{attribute 'GeneratedUsingTerminal: EK1100-0000-0018'}
{attribute addProperty BoxType "EK1100-0000-0018"}
{attribute addProperty Id "Beckhoff_EL1xxxEK1122Beckhoff_EL1xxxEK1122_A32C991B2A_0001_EL1002_0000_0000EL1002_90CA79196A_0002_EL1002_0000_0016EL1002_90CA79196A_0003_EL1002_0000_0017EL1002_90CA79196A_0004_EL1002_0000_0018EL1002_90CA79196A_0005_EL1004_0000_0000EL1004_BF8C6BFA8A_0006_EL1004_0000_0016EL1004_BF8C6BFA8A_0007_EL1004_0000_0017EL1004_BF8C6BFA8A_0008_EL1004_0000_0018EL1004_BF8C6BFA8A_0009_EL1004_0000_0019EL1004_BF8C6BFA8A_0010_EL1004_0010_0000EL1004_BF8C6BFA8A_0011_EL1004_0010_0016EL1004_BF8C6BFA8A_0012_EL1004_0010_0017EL1004_BF8C6BFA8A_0013_EL1004_0010_0018EL1004_BF8C6BFA8A_0014_EL1004_0020_0016EL1004_BF8C6BFA8A_0015_EL1008_0000_0016EL1008_4201D0AB12A_0016_EL1008_0000_0017EL1008_4201D0AB12A_0017_EL1008_0000_0018EL1008_4201D0AB12A_0018_EL1012_0000_0000EL1012_90CA79196A_0019_EL1012_0000_0016EL1012_90CA79196A_0020_EL1012_0000_0017EL1012_90CA79196A_0021_EL1012_0000_0018EL1012_90CA79196A_0022_EL1014_0000_0000EL1014_BF8C6BFA8A_0023_EL1014_0000_0016EL1014_BF8C6BFA8A_0024_EL1014_0000_0017EL1014_BF8C6BFA8A_0025_EL1014_0000_0018EL1014_BF8C6BFA8A_0026_EL1014_0000_0019EL1014_BF8C6BFA8A_0027_EL1014_0010_0000EL1014_BF8C6BFA8A_0028_EL1014_0010_0016EL1014_BF8C6BFA8A_0029_EL1014_0010_0017EL1014_BF8C6BFA8A_0030_EL1014_0010_0018EL1014_BF8C6BFA8A_0031_EL1014_0010_0019EL1014_BF8C6BFA8A_0032_EL1018_0000_0016EL1018_4201D0AB12A_0033_EL1018_0000_0017EL1018_4201D0AB12A_0034_EL1018_0000_0018EL1018_4201D0AB12A_0035_EL1024_0000_0016EL1024_BF8C6BFA8A_0036_EL1024_0000_0017EL1024_BF8C6BFA8A_0037_EL1024_0000_0018EL1024_BF8C6BFA8A_0038_EL1034_0000_0016EL1034_BF8C6BFA8A_0039_EL1034_0000_0017EL1034_BF8C6BFA8A_0040_EL1034_0000_0018EL1034_BF8C6BFA8A_0041_EL1052_0000_0016EL1052_FE4CEFB88A_0042_EL1054_0000_0016EL1054_5971E93D12A_0043_EL1084_0000_0016EL1084_BF8C6BFA8A_0044_EL1084_0000_0017EL1084_BF8C6BFA8A_0045_EL1084_0000_0018EL1084_BF8C6BFA8A_0046_EL1088_0000_0016EL1088_4201D0AB12A_0047_EL1088_0000_0017EL1088_4201D0AB12A_0048_EL1088_0000_0018EL1088_4201D0AB12A_0049_EL1094_0000_0016EL1094_BF8C6BFA8A_0050_EL1094_0000_0017EL1094_BF8C6BFA8A_0051_EL1094_0000_0018EL1094_BF8C6BFA8A_0052_EL1098_0000_0016EL1098_4201D0AB12A_0053_EL1098_0000_0017EL1098_4201D0AB12A_0054_EL1098_0000_0018EL1098_4201D0AB12A_0055_EL1104_0000_0016EL1104_BF8C6BFA8A_0056_EL1104_0000_0017EL1104_BF8C6BFA8A_0057_EL1104_0000_0018EL1104_BF8C6BFA8A_0058_EL1114_0000_0016EL1114_BF8C6BFA8A_0059_EL1114_0000_0017EL1114_BF8C6BFA8A_0060_EL1114_0000_0018EL1114_BF8C6BFA8A_0061_EL1124_0000_0016EL1124_BF8C6BFA8A_0062_EL1124_0000_0017EL1124_BF8C6BFA8A_0063_EL1124_0000_0018EL1124_BF8C6BFA8A_0064_EL1134_0000_0016EL1134_BF8C6BFA8A_0065_EL1134_0000_0017EL1134_BF8C6BFA8A_0066_EL1134_0000_0018EL1134_BF8C6BFA8A_0067_EL1144_0000_0016EL1144_BF8C6BFA8A_0068_EL1144_0000_0017EL1144_BF8C6BFA8A_0069_EL1144_0000_0018EL1144_BF8C6BFA8A_0070_EL1202_0000_0016EL1202_90CA79196A_0071_EL1202_0000_0017EL1202_90CA79196A_0072_EL1202_0000_0018EL1202_90CA79196A_0073_EL1202_0000_0019EL1202_90CA79196A_0074_EL1202_0100_0016EL1202_5869074F22A_0075_EL1202_0100_0017EL1202_5869074F22A_0076_EL1202_0100_0018EL1202_5869074F22A_0077_EL1202_0100_0019EL1202_5869074F22A_0078_EL1252_0000_0017EL1252_F879009148A_0079_EL1252_0000_0018EL1252_671E5FD948A_0080_EL1252_0000_0019EL1252_671E5FD948A_0081_EL1252_0000_0020EL1252_671E5FD948A_0082_EL1252_0000_0021EL1252_671E5FD948A_0083_EL1252_0000_0022EL1252_671E5FD948A_0084_EL1252_0010_0019EL1252_671E5FD948A_0085_EL1252_0010_0020EL1252_671E5FD948A_0086_EL1252_0010_0021EL1252_671E5FD948A_0087_EL1252_0050_0016EL1252_671E5FD948A_0088_EL1252_0050_0017EL1252_671E5FD948A_0089_EL1252_0050_0018EL1252_671E5FD948A_0090_EL1254_0000_0000EL1254_F2A8C39584A_0091_EL1262_0000_0002EL1262_BA5C56E540A_0092_EL1262_0000_0003EL1262_BA5C56E540A_0093_EL1262_0050_0002EL1262_BA5C56E540A_0094_EL1262_0050_0003EL1262_BA5C56E540A_0095_EL1258_0000_0016EL1258_D4F4E2D7484A_0096_EL1258_0000_0017EL1258_D4F4E2D7484A_0097_EL1258_0010_0017EL1258_FEC2AC79124A_0098_EL1259_0000_0016EL1259_C8DF9E9D972A_0099_EL1259_0000_0017EL1259_32A74CEC980A_0100_EL1259_0000_0018EL1259_32A74CEC980A_0101_EL1382_0000_0016EL1382_FE4CEFB88A_0102_EL1382_0000_0017EL1382_FE4CEFB88A_0103_EL1382_0000_0018EL1382_FE4CEFB88A_0104_EL1702_0000_0016EL1702_90CA79196A_0105_EL1702_0000_0017EL1702_90CA79196A_0106_EL1702_0020_0016EL1702_90CA79196A_0107_EL1712_0000_0016EL1712_90CA79196A_0108_EL1712_0020_0016EL1712_90CA79196A_0109_EL1722_0000_0016EL1722_90CA79196A_0110_EL1722_0000_0017EL1722_90CA79196A_0111_EL1804_0000_0016EL1804_BF8C6BFA8A_0112_EL1804_0000_0017EL1804_BF8C6BFA8A_0113_EL1804_0000_0018EL1804_BF8C6BFA8A_0114_EL1808_0000_0016EL1808_4201D0AB12A_0115_EL1808_0000_0017EL1808_4201D0AB12A_0116_EL1808_0000_0018EL1808_4201D0AB12A_0117_EL1809_0000_0016EL1809_FD7895E220A_0118_EL1809_0000_0017EL1809_FD7895E220A_0119_EL1809_0000_0018EL1809_FD7895E220A_0120_EL1814_0000_0016EL1814_BF8C6BFA8A_0121_EL1814_0000_0017EL1814_BF8C6BFA8A_0122_EL1814_0000_0018EL1814_BF8C6BFA8A_0123_EL1819_0000_0016EL1819_FD7895E220A_0124_EL1819_0000_0017EL1819_FD7895E220A_0125_EL1819_0000_0018EL1819_FD7895E220A_0126_EL1852_0000_0016EL1852_B9F455E920A_0127_EL1859_0000_0016EL1859_B9F455E920A_0128_EL1859_0000_0017EL1859_B9F455E920A_0129_EL1859_0000_0018EL1859_B9F455E920A_0130_EL1862_0000_0016EL1862_FD7895E220A_0131_EL1862_0000_0017EL1862_FD7895E220A_0132_EL1862_0000_0018EL1862_FD7895E220A_0133_EL1862_0000_0019EL1862_FD7895E220A_0134_EL1862_0010_0016EL1862_FD7895E220A_0135_EL1862_0010_0017EL1862_FD7895E220A_0136_EL1862_0010_0018EL1862_FD7895E220A_0137_EL1862_0010_0019EL1862_FD7895E220A_0138_EL1872_0000_0016EL1872_FD7895E220A_0139_EL1872_0000_0017EL1872_FD7895E220A_0140_EL1872_0000_0018EL1872_FD7895E220A_0141_EL1872_0010_0016EL1872_FD7895E220A_0142_EL1889_0000_0016EL1889_FD7895E220A_0143_EL1889_0000_0017EL1889_FD7895E220A_0144_EL1889_0000_0018EL1889_FD7895E220A_0145_EL1889_0000_0019EL1889_FD7895E220A_0146_EL1899_0000_0016EL1899_FD7895E220"}
{attribute addProperty CRC "3910229889"}
{attribute addProperty Size "6236"}
TYPE Beckhoff_EL1xxx_E9115F81 EXTENDS EK1100_AB5A9467 :
STRUCT
	{attribute addProperty Name "Beckhoff_EL1xxxEK1122"}
	Beckhoff_EL1xxxEK1122 : Beckhoff_EL1xxxEK1122_A32C991B;
	{attribute addProperty Name "A_0001_EL1002_0000_0000"}
	A_0001_EL1002_0000_0000 : EL1002_90CA7919;
	{attribute addProperty Name "A_0002_EL1002_0000_0016"}
	A_0002_EL1002_0000_0016 : EL1002_90CA7919;
	{attribute addProperty Name "A_0003_EL1002_0000_0017"}
	A_0003_EL1002_0000_0017 : EL1002_90CA7919;
	{attribute addProperty Name "A_0004_EL1002_0000_0018"}
	A_0004_EL1002_0000_0018 : EL1002_90CA7919;
	{attribute addProperty Name "A_0005_EL1004_0000_0000"}
	A_0005_EL1004_0000_0000 : EL1004_BF8C6BFA;
	{attribute addProperty Name "A_0006_EL1004_0000_0016"}
	A_0006_EL1004_0000_0016 : EL1004_BF8C6BFA;
	{attribute addProperty Name "A_0007_EL1004_0000_0017"}
	A_0007_EL1004_0000_0017 : EL1004_BF8C6BFA;
	{attribute addProperty Name "A_0008_EL1004_0000_0018"}
	A_0008_EL1004_0000_0018 : EL1004_BF8C6BFA;
	{attribute addProperty Name "A_0009_EL1004_0000_0019"}
	A_0009_EL1004_0000_0019 : EL1004_BF8C6BFA;
	{attribute addProperty Name "A_0010_EL1004_0010_0000"}
	A_0010_EL1004_0010_0000 : EL1004_BF8C6BFA;
	{attribute addProperty Name "A_0011_EL1004_0010_0016"}
	A_0011_EL1004_0010_0016 : EL1004_BF8C6BFA;
	{attribute addProperty Name "A_0012_EL1004_0010_0017"}
	A_0012_EL1004_0010_0017 : EL1004_BF8C6BFA;
	{attribute addProperty Name "A_0013_EL1004_0010_0018"}
	A_0013_EL1004_0010_0018 : EL1004_BF8C6BFA;
	{attribute addProperty Name "A_0014_EL1004_0020_0016"}
	A_0014_EL1004_0020_0016 : EL1004_BF8C6BFA;
	{attribute addProperty Name "A_0015_EL1008_0000_0016"}
	A_0015_EL1008_0000_0016 : EL1008_4201D0AB;
	{attribute addProperty Name "A_0016_EL1008_0000_0017"}
	A_0016_EL1008_0000_0017 : EL1008_4201D0AB;
	{attribute addProperty Name "A_0017_EL1008_0000_0018"}
	A_0017_EL1008_0000_0018 : EL1008_4201D0AB;
	{attribute addProperty Name "A_0018_EL1012_0000_0000"}
	A_0018_EL1012_0000_0000 : EL1012_90CA7919;
	{attribute addProperty Name "A_0019_EL1012_0000_0016"}
	A_0019_EL1012_0000_0016 : EL1012_90CA7919;
	{attribute addProperty Name "A_0020_EL1012_0000_0017"}
	A_0020_EL1012_0000_0017 : EL1012_90CA7919;
	{attribute addProperty Name "A_0021_EL1012_0000_0018"}
	A_0021_EL1012_0000_0018 : EL1012_90CA7919;
	{attribute addProperty Name "A_0022_EL1014_0000_0000"}
	A_0022_EL1014_0000_0000 : EL1014_BF8C6BFA;
	{attribute addProperty Name "A_0023_EL1014_0000_0016"}
	A_0023_EL1014_0000_0016 : EL1014_BF8C6BFA;
	{attribute addProperty Name "A_0024_EL1014_0000_0017"}
	A_0024_EL1014_0000_0017 : EL1014_BF8C6BFA;
	{attribute addProperty Name "A_0025_EL1014_0000_0018"}
	A_0025_EL1014_0000_0018 : EL1014_BF8C6BFA;
	{attribute addProperty Name "A_0026_EL1014_0000_0019"}
	A_0026_EL1014_0000_0019 : EL1014_BF8C6BFA;
	{attribute addProperty Name "A_0027_EL1014_0010_0000"}
	A_0027_EL1014_0010_0000 : EL1014_BF8C6BFA;
	{attribute addProperty Name "A_0028_EL1014_0010_0016"}
	A_0028_EL1014_0010_0016 : EL1014_BF8C6BFA;
	{attribute addProperty Name "A_0029_EL1014_0010_0017"}
	A_0029_EL1014_0010_0017 : EL1014_BF8C6BFA;
	{attribute addProperty Name "A_0030_EL1014_0010_0018"}
	A_0030_EL1014_0010_0018 : EL1014_BF8C6BFA;
	{attribute addProperty Name "A_0031_EL1014_0010_0019"}
	A_0031_EL1014_0010_0019 : EL1014_BF8C6BFA;
	{attribute addProperty Name "A_0032_EL1018_0000_0016"}
	A_0032_EL1018_0000_0016 : EL1018_4201D0AB;
	{attribute addProperty Name "A_0033_EL1018_0000_0017"}
	A_0033_EL1018_0000_0017 : EL1018_4201D0AB;
	{attribute addProperty Name "A_0034_EL1018_0000_0018"}
	A_0034_EL1018_0000_0018 : EL1018_4201D0AB;
	{attribute addProperty Name "A_0035_EL1024_0000_0016"}
	A_0035_EL1024_0000_0016 : EL1024_BF8C6BFA;
	{attribute addProperty Name "A_0036_EL1024_0000_0017"}
	A_0036_EL1024_0000_0017 : EL1024_BF8C6BFA;
	{attribute addProperty Name "A_0037_EL1024_0000_0018"}
	A_0037_EL1024_0000_0018 : EL1024_BF8C6BFA;
	{attribute addProperty Name "A_0038_EL1034_0000_0016"}
	A_0038_EL1034_0000_0016 : EL1034_BF8C6BFA;
	{attribute addProperty Name "A_0039_EL1034_0000_0017"}
	A_0039_EL1034_0000_0017 : EL1034_BF8C6BFA;
	{attribute addProperty Name "A_0040_EL1034_0000_0018"}
	A_0040_EL1034_0000_0018 : EL1034_BF8C6BFA;
	{attribute addProperty Name "A_0041_EL1052_0000_0016"}
	A_0041_EL1052_0000_0016 : EL1052_FE4CEFB8;
	{attribute addProperty Name "A_0042_EL1054_0000_0016"}
	A_0042_EL1054_0000_0016 : EL1054_5971E93D;
	{attribute addProperty Name "A_0043_EL1084_0000_0016"}
	A_0043_EL1084_0000_0016 : EL1084_BF8C6BFA;
	{attribute addProperty Name "A_0044_EL1084_0000_0017"}
	A_0044_EL1084_0000_0017 : EL1084_BF8C6BFA;
	{attribute addProperty Name "A_0045_EL1084_0000_0018"}
	A_0045_EL1084_0000_0018 : EL1084_BF8C6BFA;
	{attribute addProperty Name "A_0046_EL1088_0000_0016"}
	A_0046_EL1088_0000_0016 : EL1088_4201D0AB;
	{attribute addProperty Name "A_0047_EL1088_0000_0017"}
	A_0047_EL1088_0000_0017 : EL1088_4201D0AB;
	{attribute addProperty Name "A_0048_EL1088_0000_0018"}
	A_0048_EL1088_0000_0018 : EL1088_4201D0AB;
	{attribute addProperty Name "A_0049_EL1094_0000_0016"}
	A_0049_EL1094_0000_0016 : EL1094_BF8C6BFA;
	{attribute addProperty Name "A_0050_EL1094_0000_0017"}
	A_0050_EL1094_0000_0017 : EL1094_BF8C6BFA;
	{attribute addProperty Name "A_0051_EL1094_0000_0018"}
	A_0051_EL1094_0000_0018 : EL1094_BF8C6BFA;
	{attribute addProperty Name "A_0052_EL1098_0000_0016"}
	A_0052_EL1098_0000_0016 : EL1098_4201D0AB;
	{attribute addProperty Name "A_0053_EL1098_0000_0017"}
	A_0053_EL1098_0000_0017 : EL1098_4201D0AB;
	{attribute addProperty Name "A_0054_EL1098_0000_0018"}
	A_0054_EL1098_0000_0018 : EL1098_4201D0AB;
	{attribute addProperty Name "A_0055_EL1104_0000_0016"}
	A_0055_EL1104_0000_0016 : EL1104_BF8C6BFA;
	{attribute addProperty Name "A_0056_EL1104_0000_0017"}
	A_0056_EL1104_0000_0017 : EL1104_BF8C6BFA;
	{attribute addProperty Name "A_0057_EL1104_0000_0018"}
	A_0057_EL1104_0000_0018 : EL1104_BF8C6BFA;
	{attribute addProperty Name "A_0058_EL1114_0000_0016"}
	A_0058_EL1114_0000_0016 : EL1114_BF8C6BFA;
	{attribute addProperty Name "A_0059_EL1114_0000_0017"}
	A_0059_EL1114_0000_0017 : EL1114_BF8C6BFA;
	{attribute addProperty Name "A_0060_EL1114_0000_0018"}
	A_0060_EL1114_0000_0018 : EL1114_BF8C6BFA;
	{attribute addProperty Name "A_0061_EL1124_0000_0016"}
	A_0061_EL1124_0000_0016 : EL1124_BF8C6BFA;
	{attribute addProperty Name "A_0062_EL1124_0000_0017"}
	A_0062_EL1124_0000_0017 : EL1124_BF8C6BFA;
	{attribute addProperty Name "A_0063_EL1124_0000_0018"}
	A_0063_EL1124_0000_0018 : EL1124_BF8C6BFA;
	{attribute addProperty Name "A_0064_EL1134_0000_0016"}
	A_0064_EL1134_0000_0016 : EL1134_BF8C6BFA;
	{attribute addProperty Name "A_0065_EL1134_0000_0017"}
	A_0065_EL1134_0000_0017 : EL1134_BF8C6BFA;
	{attribute addProperty Name "A_0066_EL1134_0000_0018"}
	A_0066_EL1134_0000_0018 : EL1134_BF8C6BFA;
	{attribute addProperty Name "A_0067_EL1144_0000_0016"}
	A_0067_EL1144_0000_0016 : EL1144_BF8C6BFA;
	{attribute addProperty Name "A_0068_EL1144_0000_0017"}
	A_0068_EL1144_0000_0017 : EL1144_BF8C6BFA;
	{attribute addProperty Name "A_0069_EL1144_0000_0018"}
	A_0069_EL1144_0000_0018 : EL1144_BF8C6BFA;
	{attribute addProperty Name "A_0070_EL1202_0000_0016"}
	A_0070_EL1202_0000_0016 : EL1202_90CA7919;
	{attribute addProperty Name "A_0071_EL1202_0000_0017"}
	A_0071_EL1202_0000_0017 : EL1202_90CA7919;
	{attribute addProperty Name "A_0072_EL1202_0000_0018"}
	A_0072_EL1202_0000_0018 : EL1202_90CA7919;
	{attribute addProperty Name "A_0073_EL1202_0000_0019"}
	A_0073_EL1202_0000_0019 : EL1202_90CA7919;
	{attribute addProperty Name "A_0074_EL1202_0100_0016"}
	A_0074_EL1202_0100_0016 : EL1202_5869074F;
	{attribute addProperty Name "A_0075_EL1202_0100_0017"}
	A_0075_EL1202_0100_0017 : EL1202_5869074F;
	{attribute addProperty Name "A_0076_EL1202_0100_0018"}
	A_0076_EL1202_0100_0018 : EL1202_5869074F;
	{attribute addProperty Name "A_0077_EL1202_0100_0019"}
	A_0077_EL1202_0100_0019 : EL1202_5869074F;
	{attribute addProperty Name "A_0078_EL1252_0000_0017"}
	A_0078_EL1252_0000_0017 : EL1252_F8790091;
	{attribute addProperty Name "A_0079_EL1252_0000_0018"}
	A_0079_EL1252_0000_0018 : EL1252_671E5FD9;
	{attribute addProperty Name "A_0080_EL1252_0000_0019"}
	A_0080_EL1252_0000_0019 : EL1252_671E5FD9;
	{attribute addProperty Name "A_0081_EL1252_0000_0020"}
	A_0081_EL1252_0000_0020 : EL1252_671E5FD9;
	{attribute addProperty Name "A_0082_EL1252_0000_0021"}
	A_0082_EL1252_0000_0021 : EL1252_671E5FD9;
	{attribute addProperty Name "A_0083_EL1252_0000_0022"}
	A_0083_EL1252_0000_0022 : EL1252_671E5FD9;
	{attribute addProperty Name "A_0084_EL1252_0010_0019"}
	A_0084_EL1252_0010_0019 : EL1252_671E5FD9;
	{attribute addProperty Name "A_0085_EL1252_0010_0020"}
	A_0085_EL1252_0010_0020 : EL1252_671E5FD9;
	{attribute addProperty Name "A_0086_EL1252_0010_0021"}
	A_0086_EL1252_0010_0021 : EL1252_671E5FD9;
	{attribute addProperty Name "A_0087_EL1252_0050_0016"}
	A_0087_EL1252_0050_0016 : EL1252_671E5FD9;
	{attribute addProperty Name "A_0088_EL1252_0050_0017"}
	A_0088_EL1252_0050_0017 : EL1252_671E5FD9;
	{attribute addProperty Name "A_0089_EL1252_0050_0018"}
	A_0089_EL1252_0050_0018 : EL1252_671E5FD9;
	{attribute addProperty Name "A_0090_EL1254_0000_0000"}
	A_0090_EL1254_0000_0000 : EL1254_F2A8C395;
	{attribute addProperty Name "A_0091_EL1262_0000_0002"}
	A_0091_EL1262_0000_0002 : EL1262_BA5C56E5;
	{attribute addProperty Name "A_0092_EL1262_0000_0003"}
	A_0092_EL1262_0000_0003 : EL1262_BA5C56E5;
	{attribute addProperty Name "A_0093_EL1262_0050_0002"}
	A_0093_EL1262_0050_0002 : EL1262_BA5C56E5;
	{attribute addProperty Name "A_0094_EL1262_0050_0003"}
	A_0094_EL1262_0050_0003 : EL1262_BA5C56E5;
	{attribute addProperty Name "A_0095_EL1258_0000_0016"}
	A_0095_EL1258_0000_0016 : EL1258_D4F4E2D7;
	{attribute addProperty Name "A_0096_EL1258_0000_0017"}
	A_0096_EL1258_0000_0017 : EL1258_D4F4E2D7;
	{attribute addProperty Name "A_0097_EL1258_0010_0017"}
	A_0097_EL1258_0010_0017 : EL1258_FEC2AC79;
	{attribute addProperty Name "A_0098_EL1259_0000_0016"}
	A_0098_EL1259_0000_0016 : EL1259_C8DF9E9D;
	{attribute addProperty Name "A_0099_EL1259_0000_0017"}
	A_0099_EL1259_0000_0017 : EL1259_32A74CEC;
	{attribute addProperty Name "A_0100_EL1259_0000_0018"}
	A_0100_EL1259_0000_0018 : EL1259_32A74CEC;
	{attribute addProperty Name "A_0101_EL1382_0000_0016"}
	A_0101_EL1382_0000_0016 : EL1382_FE4CEFB8;
	{attribute addProperty Name "A_0102_EL1382_0000_0017"}
	A_0102_EL1382_0000_0017 : EL1382_FE4CEFB8;
	{attribute addProperty Name "A_0103_EL1382_0000_0018"}
	A_0103_EL1382_0000_0018 : EL1382_FE4CEFB8;
	{attribute addProperty Name "A_0104_EL1702_0000_0016"}
	A_0104_EL1702_0000_0016 : EL1702_90CA7919;
	{attribute addProperty Name "A_0105_EL1702_0000_0017"}
	A_0105_EL1702_0000_0017 : EL1702_90CA7919;
	{attribute addProperty Name "A_0106_EL1702_0020_0016"}
	A_0106_EL1702_0020_0016 : EL1702_90CA7919;
	{attribute addProperty Name "A_0107_EL1712_0000_0016"}
	A_0107_EL1712_0000_0016 : EL1712_90CA7919;
	{attribute addProperty Name "A_0108_EL1712_0020_0016"}
	A_0108_EL1712_0020_0016 : EL1712_90CA7919;
	{attribute addProperty Name "A_0109_EL1722_0000_0016"}
	A_0109_EL1722_0000_0016 : EL1722_90CA7919;
	{attribute addProperty Name "A_0110_EL1722_0000_0017"}
	A_0110_EL1722_0000_0017 : EL1722_90CA7919;
	{attribute addProperty Name "A_0111_EL1804_0000_0016"}
	A_0111_EL1804_0000_0016 : EL1804_BF8C6BFA;
	{attribute addProperty Name "A_0112_EL1804_0000_0017"}
	A_0112_EL1804_0000_0017 : EL1804_BF8C6BFA;
	{attribute addProperty Name "A_0113_EL1804_0000_0018"}
	A_0113_EL1804_0000_0018 : EL1804_BF8C6BFA;
	{attribute addProperty Name "A_0114_EL1808_0000_0016"}
	A_0114_EL1808_0000_0016 : EL1808_4201D0AB;
	{attribute addProperty Name "A_0115_EL1808_0000_0017"}
	A_0115_EL1808_0000_0017 : EL1808_4201D0AB;
	{attribute addProperty Name "A_0116_EL1808_0000_0018"}
	A_0116_EL1808_0000_0018 : EL1808_4201D0AB;
	{attribute addProperty Name "A_0117_EL1809_0000_0016"}
	A_0117_EL1809_0000_0016 : EL1809_FD7895E2;
	{attribute addProperty Name "A_0118_EL1809_0000_0017"}
	A_0118_EL1809_0000_0017 : EL1809_FD7895E2;
	{attribute addProperty Name "A_0119_EL1809_0000_0018"}
	A_0119_EL1809_0000_0018 : EL1809_FD7895E2;
	{attribute addProperty Name "A_0120_EL1814_0000_0016"}
	A_0120_EL1814_0000_0016 : EL1814_BF8C6BFA;
	{attribute addProperty Name "A_0121_EL1814_0000_0017"}
	A_0121_EL1814_0000_0017 : EL1814_BF8C6BFA;
	{attribute addProperty Name "A_0122_EL1814_0000_0018"}
	A_0122_EL1814_0000_0018 : EL1814_BF8C6BFA;
	{attribute addProperty Name "A_0123_EL1819_0000_0016"}
	A_0123_EL1819_0000_0016 : EL1819_FD7895E2;
	{attribute addProperty Name "A_0124_EL1819_0000_0017"}
	A_0124_EL1819_0000_0017 : EL1819_FD7895E2;
	{attribute addProperty Name "A_0125_EL1819_0000_0018"}
	A_0125_EL1819_0000_0018 : EL1819_FD7895E2;
	{attribute addProperty Name "A_0126_EL1852_0000_0016"}
	A_0126_EL1852_0000_0016 : EL1852_B9F455E9;
	{attribute addProperty Name "A_0127_EL1859_0000_0016"}
	A_0127_EL1859_0000_0016 : EL1859_B9F455E9;
	{attribute addProperty Name "A_0128_EL1859_0000_0017"}
	A_0128_EL1859_0000_0017 : EL1859_B9F455E9;
	{attribute addProperty Name "A_0129_EL1859_0000_0018"}
	A_0129_EL1859_0000_0018 : EL1859_B9F455E9;
	{attribute addProperty Name "A_0130_EL1862_0000_0016"}
	A_0130_EL1862_0000_0016 : EL1862_FD7895E2;
	{attribute addProperty Name "A_0131_EL1862_0000_0017"}
	A_0131_EL1862_0000_0017 : EL1862_FD7895E2;
	{attribute addProperty Name "A_0132_EL1862_0000_0018"}
	A_0132_EL1862_0000_0018 : EL1862_FD7895E2;
	{attribute addProperty Name "A_0133_EL1862_0000_0019"}
	A_0133_EL1862_0000_0019 : EL1862_FD7895E2;
	{attribute addProperty Name "A_0134_EL1862_0010_0016"}
	A_0134_EL1862_0010_0016 : EL1862_FD7895E2;
	{attribute addProperty Name "A_0135_EL1862_0010_0017"}
	A_0135_EL1862_0010_0017 : EL1862_FD7895E2;
	{attribute addProperty Name "A_0136_EL1862_0010_0018"}
	A_0136_EL1862_0010_0018 : EL1862_FD7895E2;
	{attribute addProperty Name "A_0137_EL1862_0010_0019"}
	A_0137_EL1862_0010_0019 : EL1862_FD7895E2;
	{attribute addProperty Name "A_0138_EL1872_0000_0016"}
	A_0138_EL1872_0000_0016 : EL1872_FD7895E2;
	{attribute addProperty Name "A_0139_EL1872_0000_0017"}
	A_0139_EL1872_0000_0017 : EL1872_FD7895E2;
	{attribute addProperty Name "A_0140_EL1872_0000_0018"}
	A_0140_EL1872_0000_0018 : EL1872_FD7895E2;
	{attribute addProperty Name "A_0141_EL1872_0010_0016"}
	A_0141_EL1872_0010_0016 : EL1872_FD7895E2;
	{attribute addProperty Name "A_0142_EL1889_0000_0016"}
	A_0142_EL1889_0000_0016 : EL1889_FD7895E2;
	{attribute addProperty Name "A_0143_EL1889_0000_0017"}
	A_0143_EL1889_0000_0017 : EL1889_FD7895E2;
	{attribute addProperty Name "A_0144_EL1889_0000_0018"}
	A_0144_EL1889_0000_0018 : EL1889_FD7895E2;
	{attribute addProperty Name "A_0145_EL1889_0000_0019"}
	A_0145_EL1889_0000_0019 : EL1889_FD7895E2;
	{attribute addProperty Name "A_0146_EL1899_0000_0016"}
	A_0146_EL1899_0000_0016 : EL1899_FD7895E2;
END_STRUCT
END_TYPE

(* stored: Version 1.2.0.0, ProductVersion 3.1.4024.9
   DUT Beckhoff_EL1xxx_E9115F81: Id {a45694a3-2676-4289-b6ea-febfc90cd4d5} *)
